% RSLogix 500 project Timers.RSS, saved by version 8.30.00.16 %
PROJECT "LEC23"    % processor: Bul.1763 MicroLogix 1100 Series B %

PROGRAM FILES
  LAD 2   14 rungs

DATA FILES
  O0 OUTPUT  4 elements
  I1 INPUT  6 elements
  S2 STATUS  66 elements
  B3 BINARY  1 elements
  T4 TIMER  3 elements
  C5 COUNTER  1 elements
  R6 CONTROL  1 elements
  N7 INTEGER  1 elements
  F8 FLOAT  1 elements

LADDER 2
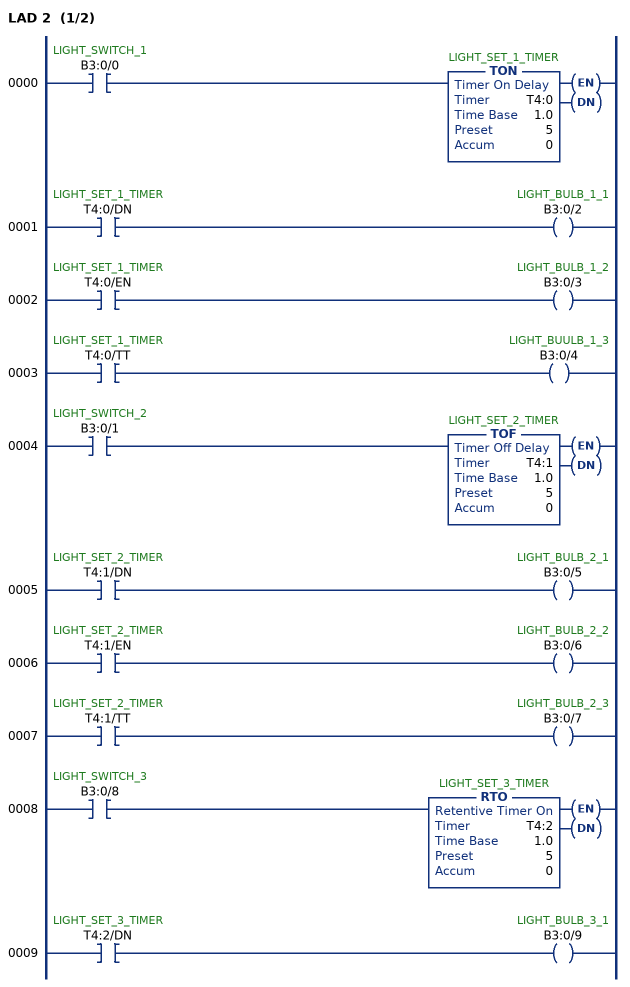
% Rung: 0 %
SOR XIC B3:0/0 TON T4:0 1.0 5 0 EOR
%   B3:0/0  "LIGHT_SWITCH_1" %
%   T4:0  "LIGHT_SET_1_TIMER" %
% Rung: 1 %
SOR XIC T4:0/DN OTE B3:0/2 EOR
%   T4:0/DN  "LIGHT_SET_1_TIMER" %
%   B3:0/2  "LIGHT_BULB_1_1" %
% Rung: 2 %
SOR XIC T4:0/EN OTE B3:0/3 EOR
%   T4:0/EN  "LIGHT_SET_1_TIMER" %
%   B3:0/3  "LIGHT_BULB_1_2" %
% Rung: 3 %
SOR XIC T4:0/TT OTE B3:0/4 EOR
%   T4:0/TT  "LIGHT_SET_1_TIMER" %
%   B3:0/4  "LIGHT_BUULB_1_3" %
% Rung: 4 %
SOR XIC B3:0/1 TOF T4:1 1.0 5 0 EOR
%   B3:0/1  "LIGHT_SWITCH_2" %
%   T4:1  "LIGHT_SET_2_TIMER" %
% Rung: 5 %
SOR XIC T4:1/DN OTE B3:0/5 EOR
%   T4:1/DN  "LIGHT_SET_2_TIMER" %
%   B3:0/5  "LIGHT_BULB_2_1" %
% Rung: 6 %
SOR XIC T4:1/EN OTE B3:0/6 EOR
%   T4:1/EN  "LIGHT_SET_2_TIMER" %
%   B3:0/6  "LIGHT_BULB_2_2" %
% Rung: 7 %
SOR XIC T4:1/TT OTE B3:0/7 EOR
%   T4:1/TT  "LIGHT_SET_2_TIMER" %
%   B3:0/7  "LIGHT_BULB_2_3" %
% Rung: 8 %
SOR XIC B3:0/8 RTO T4:2 1.0 5 0 EOR
%   B3:0/8  "LIGHT_SWITCH_3" %
%   T4:2  "LIGHT_SET_3_TIMER" %
% Rung: 9 %
SOR XIC T4:2/DN OTE B3:0/9 EOR
%   T4:2/DN  "LIGHT_SET_3_TIMER" %
%   B3:0/9  "LIGHT_BULB_3_1" %

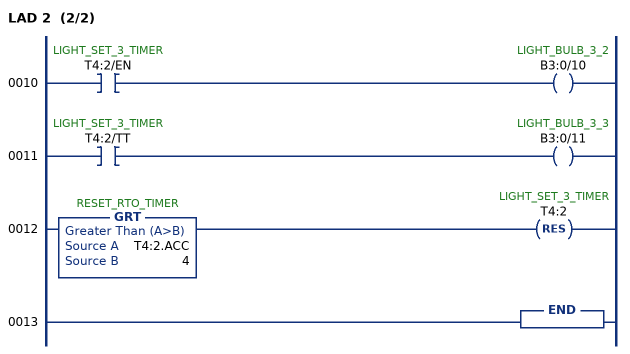
% Rung: 10 %
SOR XIC T4:2/EN OTE B3:0/10 EOR
%   T4:2/EN  "LIGHT_SET_3_TIMER" %
%   B3:0/10  "LIGHT_BULB_3_2" %
% Rung: 11 %
SOR XIC T4:2/TT OTE B3:0/11 EOR
%   T4:2/TT  "LIGHT_SET_3_TIMER" %
%   B3:0/11  "LIGHT_BULB_3_3" %
% Rung: 12 %
SOR GRT T4:2.ACC 4 RES T4:2 EOR
%   T4:2.ACC  "RESET_RTO_TIMER" %
%   T4:2  "LIGHT_SET_3_TIMER" %
% Rung: 13 %
SOR END EOR

OTHER DOCUMENTED ADDRESSES
  T4:3/DN  "LIGHT_SET_3_TIMER"
  T4:3/TT  "LIGHT_SET_3_TIMER"

REVISION NOTES
  0: Changed RTO
  1: Added comparison for reset

DATA TABLE (non-zero values as saved)
DATA T4
% .PRE .ACC %
% T4:0 % 5 0
% T4:1 % 5 0
% T4:2 % 5 0
